# B&R Automation Studio project Snapshot (part 2)

#### Function Description1.txt
```
===================================================================================#
This is a sample trak project for the purposes of testing out the snapshot feature.#
===================================================================================#
Function:                                                                          #
50 shuttles move around the trak to move a product from station to station. This   #
continues until the product is finished and unloaded or rejected and removed.      #
                                                                                   #
                                                                                   #
Production stages:                                                                 #
The product can exist in four different states. At each stage, the product becomes #
harder/firmer and can be moved faster and accelerated quicker. The four stages and #
their respective parameters are:                                                   #
                                                                                   #
1 YELLOW (Liquid)                                                                  #
	veloctiy    = 0.5 m/s                                                          #
	accel/decel = 5 m/s^2                                                          #
	destination = stn 2                                                            #
2 BLUE (Gel)                                                                       #
	veloctiy    = 1 m/s                                                            #
	accel/decel = 10 m/s^2                                                         #
	destination = stn 3                                                            #
3 ORANGE (Soft Solid)                                                              #
	veloctiy    = 2 m/s                                                            #
	accel/decel = 15 m/s^2                                                         #
	destination = stn 4                                                            #
4 GREEN (Solid)                                                                    #
	veloctiy    = 2.5 m/s                                                          #
	accel/decel = 20 m/s^2                                                         #
	destination = stn 1 (offload)                                                  #
                                                                                   #
                                                                                   #
Additional stages:                                                                 #
The two additional stages are:                                                     #
                                                                                   #
1 GRAY (Empty Shuttle)                                                             #
	veloctiy    = 4 m/s                                                            #
	accel/decel = 20 m/s^2                                                         #
	destination = stn 1                                                            #
2 RED (Rejected Product)                                                           #
	veloctiy    = retains speed based on matter state                              #
	accel/decel = retains accel/decel based on matter state                        #
	destination = stn 5 (liquids and gels) or stn 6 (Soft Solids and Solids)       #
                                                                                   #
                                                                                   #
Station Descriptions:                                                              #
                                                                                   #
1 Load/Unload                                                                      #
	Empty shuttles recieve a liquid product                                        #
	GRAY -> YELLOW                                                                 #
	Goes to stn 2                                                                  #
	Finished solid products are removed and the empty shuttles are sent around     #
	GREEN -> GREY                                                                  #
	Goes to stn 1                                                                  #
2 Process 1                                                                        #
	Liquid products are made into gels                                             #
	YELLOW -> BLUE                                                                 #
	Goes to stn 3                                                                  #
3 Process 2                                                                        #
	Gel products are made into soft solids                                         #
	BLUE -> ORANGE                                                                 #
	Goes to stn 4                                                                  #
4 Process 3                                                                        #
	Soft solid products are made into solids                                       #
	ORANGE -> GREEN                                                                #
	Goes to stn 1                                                                  #
5 Reject 1                                                                         #
	Rejected liquid and gel products are removed                                   #
	RED -> GRAY                                                                    #
	Goes to stn 1                                                                  #
6 Reject 2                                                                         #
	Rejected soft solid and solid products are removed                             #
	RED -> GREY                                                                    #
	Goes to stn 1                                                                  #
                                                                                   #
                                                                                   #
At random times, stations will detect rejects, turn them red, and send them to the #
appropriate reject stations.                                                       #
===================================================================================#
```

#### Init.st
```iecst
PROGRAM _INIT
	//Build the array of station references
	Stn[1]  := ADR(Load_Unload_Sector);

	Stn[2]  := ADR(Process_1_Sector);

	Stn[3]  := ADR(Process_2_Sector);

	Stn[4]  := ADR(Process_3_Sector);

	Stn[5]  := ADR(Reject_LeftUp);
	Stn[6]  := ADR(Reject_RightUp);
	Stn[7]  := ADR(Reject_RightDown);

	Stn[8]  := ADR(Flipper_LeftUp);
	Stn[9]  := ADR(Flipper_RightUp);
	Stn[10] := ADR(Flipper_RightDown);

	//List the segment sectors
	SECTOR_SEG_01;
	SECTOR_SEG_02;
	SECTOR_SEG_03;
	SECTOR_SEG_04;
	SECTOR_SEG_05;
	SECTOR_SEG_06;
	SECTOR_SEG_07;
	SECTOR_SEG_08;
	SECTOR_SEG_09;
	SECTOR_SEG_10;
	SECTOR_SEG_11;
	SECTOR_SEG_12;
	SECTOR_SEG_13;
	SECTOR_SEG_14;
	SECTOR_SEG_15;
	SECTOR_SEG_16;
	SECTOR_SEG_17;
	SECTOR_SEG_18;
	SECTOR_SEG_19;
	SECTOR_SEG_20;
	SECTOR_SEG_21;
	SECTOR_SEG_22;
	SECTOR_SEG_23;
	SECTOR_SEG_24;
	SECTOR_SEG_25;
	SECTOR_SEG_26;
	SECTOR_SEG_27;
	SECTOR_SEG_28;
	SECTOR_SEG_29;
	SECTOR_SEG_30;
	SECTOR_SEG_31;
	SECTOR_SEG_32;
	SECTOR_SEG_33;
	SECTOR_SEG_34;
	SECTOR_SEG_35;
	SECTOR_SEG_36;
	SECTOR_SEG_37;
	SECTOR_SEG_38;
	SECTOR_SEG_39;
	SECTOR_SEG_40;
	SECTOR_SEG_41;
	SECTOR_SEG_42;
	SECTOR_SEG_43;
	SECTOR_SEG_44;
	SECTOR_SEG_45;
	SECTOR_SEG_46;
	SECTOR_SEG_47;
	SECTOR_SEG_48;
	SECTOR_SEG_49;
	SECTOR_SEG_50;
	SECTOR_SEG_51;
	SECTOR_SEG_52;
	SECTOR_SEG_53;
	SECTOR_SEG_54;
	SECTOR_SEG_55;
	SECTOR_SEG_56;
	SECTOR_SEG_57;
	SECTOR_SEG_58;
	SECTOR_SEG_59;
	SECTOR_SEG_60;
	SECTOR_SEG_61;
	SECTOR_SEG_62;
	SECTOR_SEG_63;
	SECTOR_SEG_64;
	SECTOR_SEG_65;
	SECTOR_SEG_66;
	SECTOR_SEG_67;
	SECTOR_SEG_68;
	SECTOR_SEG_69;
	SECTOR_SEG_70;
END_PROGRAM
```

#### Main.st
```iecst
PROGRAM _CYCLIC

	BarrierReadInfo.ProcessPoint := ADR(PP_RejectEntrance);
	BarrierReadInfo.Enable       := TRUE;
	BarrierReadInfo();

	CASE TrakState OF
		TRAK_IDLE:
			IF gPowerOn THEN
				AsmPowerOn.Assembly := ADR(gAssembly_1);
				AsmPowerOn.Execute  := TRUE;
				TrakState           := TRAK_POWERON;
			END_IF

		TRAK_POWERON:
			IF AsmPowerOn.Done THEN
				AsmGetShuttle.Assembly := ADR(gAssembly_1);
				AsmGetShuttle.Enable   := TRUE;
				TrakState              := TRAK_FIND_SHUTTLE;   //USE THIS FOR REGULAR OPERATION
//				TrakState              := TRAK_SYSTEM_RUNNING; //USE THIS FOR SPAWNING OPERATION
			END_IF

		TRAK_FIND_SHUTTLE:
			IF AsmGetShuttle.Valid THEN
				AsmData.Color                 := GRAY;
				AsmCopyUserData.Axis          := ADR(AsmGetShuttle.Axis);
				AsmCopyUserData.DataAddress   := ADR(AsmData);
				AsmCopyUserData.DataSize      := SIZEOF(AsmData);
				AsmCopyUserData.Mode          := mcACPTRAK_USERDATA_SET;
				AsmCopyUserData.Execute       := TRUE;

				AsmGetShuttle.Next            := FALSE;
				AsmRoutedMoveAbs.Axis         := ADR(AsmGetShuttle.Axis);
				AsmRoutedMoveAbs.Sector       := Stn[1];
				AsmRoutedMoveAbs.Position     := 0.005;
				AsmRoutedMoveAbs.Acceleration := 20;
				AsmRoutedMoveAbs.Deceleration := 20;
				AsmRoutedMoveAbs.Velocity     := 4;
				AsmRoutedMoveAbs.Execute      := TRUE;

				TrakState                     := TRAK_SEND_SHUTTLE;
			END_IF

		TRAK_SEND_SHUTTLE:
			IF AsmRoutedMoveAbs.Active AND AsmCopyUserData.Done THEN
				IF (AsmGetShuttle.RemainingCount > 0) THEN
					AsmCopyUserData.Execute  := FALSE;
					AsmRoutedMoveAbs.Execute := FALSE;
					AsmGetShuttle.Next       := TRUE;
					//AsmIndex               := AsmIndex + 1;
					TrakState                := TRAK_FIND_SHUTTLE;
				ELSE
					AsmGetShuttle.Enable := FALSE;
					gTrakRunning         := TRUE;
					TrakState            := TRAK_SYSTEM_RUNNING;
				END_IF
			END_IF

		TRAK_SYSTEM_RUNNING:

	END_CASE

	//Call FUBs
	AsmPowerOn();
	AsmGetShuttle();
	AsmCopyUserData();
	AsmRoutedMoveAbs();

	//Call action files
	Load_Unload;
	Process_1;
	Process_2;
	Process_3;
	Reject;
	RejectExit;
	Flipper;
	FlipperExit;

END_PROGRAM
```

#### 1_Load_Unload.st
```iecst
ACTION Load_Unload:

	TrgPointEnable[1].ProcessPoint  := ADR(PP_Load_Unload);
	TrgPointEnable[1].Enable        := TRUE;
	TrgPointGetInfo[1].ProcessPoint := ADR(PP_Load_Unload);

	CASE StnState[1] OF
		STN_WAIT_FOR_SHUTTLE:
			IF (TrgPointEnable[1].EventCount > 0) THEN
				TrgPointGetInfo[1].Execute := TRUE;
				StnState[1]                := STN_GET_INFO;
			END_IF

		STN_GET_INFO:
			IF TrgPointGetInfo[1].Done THEN
				ShCopyUserData[1].Axis        := ADR(TrgPointGetInfo[1].TrgPointInfo.Axis);
				ShCopyUserData[1].DataAddress := ADR(StationData[1]);
				ShCopyUserData[1].DataSize    := SIZEOF(StationData[1]);
				ShCopyUserData[1].Mode        := mcACPTRAK_USERDATA_GET;
				ShCopyUserData[1].Execute     := TRUE;
				StnState[1]                   := STN_GET_USERDATA;
			END_IF

		STN_GET_USERDATA:
			IF ShCopyUserData[1].Done THEN
				ShCopyUserData[1].Execute := FALSE;
				IF (StationData[1].Color = GRAY) OR (StationData[1].Color = GREEN) THEN
					StnState[1] := STN_HANDLE_SHUTTLE;
				ELSE
					TrgPointGetInfo[1].Execute := FALSE;
					StnState[1]                := STN_WAIT_FOR_SHUTTLE;
				END_IF
			END_IF

		STN_HANDLE_SHUTTLE:
			IF (StationData[1].Color = GRAY) THEN
				StationData[1].Color                                      := YELLOW;
				StnRoutedMoveAbs[1].Axis                                  := ADR(TrgPointGetInfo[1].TrgPointInfo.Axis);
				StnRoutedMoveAbs[1].Sector                                := Stn[2];
				StnRoutedMoveAbs[1].Position                              := 0.005;
				StnRoutedMoveAbs[1].Acceleration                          := 5;
				StnRoutedMoveAbs[1].Deceleration                          := 5;
				StnRoutedMoveAbs[1].Velocity                              := 0.5;
				StnRoutedMoveAbs[5].AdvancedParameters.ShuttleOrientation := mcDIR_UNDEFINED;
				StnRoutedMoveAbs[1].AdvancedParameters.StartDirection     := mcDIR_POSITIVE;
				StnRoutedMoveAbs[1].AdvancedParameters.EndDirection       := mcDIR_POSITIVE;
			ELSIF (StationData[1].Color = GREEN) THEN
				IF (RejectIndex[1] = RejectRate) THEN
					StationData[1].Color                                      := RED;
					StnRoutedMoveAbs[1].Axis                                  := ADR(TrgPointGetInfo[1].TrgPointInfo.Axis);
					StnRoutedMoveAbs[1].Sector                                := Stn[6];
					StnRoutedMoveAbs[1].Position                              := 0.405;
					StnRoutedMoveAbs[1].Acceleration                          := 20;
					StnRoutedMoveAbs[1].Deceleration                          := 20;
					StnRoutedMoveAbs[1].Velocity                              := 2.5;
					StnRoutedMoveAbs[1].AdvancedParameters.ShuttleOrientation := mcDIR_UNDEFINED;
					StnRoutedMoveAbs[1].AdvancedParameters.StartDirection     := mcDIR_POSITIVE;
					StnRoutedMoveAbs[1].AdvancedParameters.EndDirection       := mcDIR_POSITIVE;
					RejectIndex[1]                                            := 0;
				ELSE
					StationData[1].Color := GRAY;
					StnRoutedMoveAbs[1].Axis                                  := ADR(TrgPointGetInfo[1].TrgPointInfo.Axis);
					StnRoutedMoveAbs[1].Sector                                := Stn[1];
					StnRoutedMoveAbs[1].Position                              := 0.004;
					StnRoutedMoveAbs[1].Acceleration                          := 20;
					StnRoutedMoveAbs[1].Deceleration                          := 20;
					StnRoutedMoveAbs[1].Velocity                              := 4;
					StnRoutedMoveAbs[5].AdvancedParameters.ShuttleOrientation := mcDIR_UNDEFINED;
					StnRoutedMoveAbs[1].AdvancedParameters.StartDirection     := mcDIR_POSITIVE;
					StnRoutedMoveAbs[1].AdvancedParameters.EndDirection       := mcDIR_POSITIVE;
					RejectIndex[1]                                            := RejectIndex[1] + 1;
				END_IF
			END_IF
			ShCopyUserData[1].Mode    := mcACPTRAK_USERDATA_SET;
			ShCopyUserData[1].Execute := TRUE;
			StnState[1]               := STN_SET_USERDATA;

		STN_SET_USERDATA:
			IF ShCopyUserData[1].Done THEN
				ShCopyUserData[1].Execute   := FALSE;
				StnRoutedMoveAbs[1].Execute := TRUE;
				StnState[1]                 := STN_SEND_SHUTTLE;
			END_IF

		STN_SEND_SHUTTLE:
			IF StnRoutedMoveAbs[1].Active THEN
				TrgPointGetInfo[1].Execute  := FALSE;
				StnRoutedMoveAbs[1].Execute := FALSE;
				StnState[1]                 := STN_WAIT_FOR_SHUTTLE;
			END_IF

	END_CASE

	TrgPointEnable[1]();
	TrgPointGetInfo[1]();
	ShCopyUserData[1]();
	StnRoutedMoveAbs[1]();

END_ACTION
```

#### 2_Process_1.st
```iecst
ACTION Process_1:

	TrgPointEnable[2].ProcessPoint  := ADR(PP_Process_1);
	TrgPointEnable[2].Enable        := TRUE;
	TrgPointGetInfo[2].ProcessPoint := ADR(PP_Process_1);

	CASE StnState[2] OF
		STN_WAIT_FOR_SHUTTLE:
			IF (TrgPointEnable[2].EventCount > 0) THEN
				TrgPointGetInfo[2].Execute := TRUE;
				StnState[2]                := STN_GET_INFO;
			END_IF

		STN_GET_INFO:
			IF TrgPointGetInfo[2].Done THEN
				ShCopyUserData[2].Axis        := ADR(TrgPointGetInfo[2].TrgPointInfo.Axis);
				ShCopyUserData[2].DataAddress := ADR(StationData[2]);
				ShCopyUserData[2].DataSize    := SIZEOF(StationData[2]);
				ShCopyUserData[2].Mode        := mcACPTRAK_USERDATA_GET;
				ShCopyUserData[2].Execute     := TRUE;
				StnState[2]                   := STN_GET_USERDATA;
			END_IF

		STN_GET_USERDATA:
			IF ShCopyUserData[2].Done THEN
				ShCopyUserData[2].Execute := FALSE;
				IF (StationData[2].Color = YELLOW) THEN
					StnState[2] := STN_HANDLE_SHUTTLE;
				ELSE
					TrgPointGetInfo[2].Execute := FALSE;
					StnState[2]                := STN_WAIT_FOR_SHUTTLE;
				END_IF
			END_IF

		STN_HANDLE_SHUTTLE:
			IF (StationData[2].Color = YELLOW) THEN
				IF (RejectIndex[2] = RejectRate) THEN
					StationData[2].Color                                      := RED;
					StnRoutedMoveAbs[2].Axis                                  := ADR(TrgPointGetInfo[2].TrgPointInfo.Axis);
					StnRoutedMoveAbs[2].Sector                                := Stn[6];
					StnRoutedMoveAbs[2].Position                              := 0.405;
					StnRoutedMoveAbs[2].Acceleration                          := 5;
					StnRoutedMoveAbs[2].Deceleration                          := 5;
					StnRoutedMoveAbs[2].Velocity                              := 0.5;
					StnRoutedMoveAbs[5].AdvancedParameters.ShuttleOrientation := mcDIR_UNDEFINED;
					StnRoutedMoveAbs[2].AdvancedParameters.StartDirection     := mcDIR_POSITIVE;
					StnRoutedMoveAbs[2].AdvancedParameters.EndDirection       := mcDIR_POSITIVE;
					RejectIndex[2]                                            := 0;
				ELSE
					StationData[2].Color                                      := BLUE;
					StnRoutedMoveAbs[2].Axis                                  := ADR(TrgPointGetInfo[2].TrgPointInfo.Axis);
					StnRoutedMoveAbs[2].Sector                                := Stn[3];
					StnRoutedMoveAbs[2].Position                              := 0.005;
					StnRoutedMoveAbs[2].Acceleration                          := 10;
					StnRoutedMoveAbs[2].Deceleration                          := 10;
					StnRoutedMoveAbs[2].Velocity                              := 1;
					StnRoutedMoveAbs[5].AdvancedParameters.ShuttleOrientation := mcDIR_UNDEFINED;
					StnRoutedMoveAbs[2].AdvancedParameters.StartDirection     := mcDIR_POSITIVE;
					StnRoutedMoveAbs[2].AdvancedParameters.EndDirection       := mcDIR_POSITIVE;
					RejectIndex[2]                                            := RejectIndex[2] + 1;
				END_IF
			END_IF
			ShCopyUserData[2].Mode    := mcACPTRAK_USERDATA_SET;
			ShCopyUserData[2].Execute := TRUE;
			StnState[2]               := STN_SET_USERDATA;

		STN_SET_USERDATA:
			IF ShCopyUserData[2].Done THEN
				ShCopyUserData[2].Execute   := FALSE;
				StnRoutedMoveAbs[2].Execute := TRUE;
				StnState[2]                 := STN_SEND_SHUTTLE;
			END_IF

		STN_SEND_SHUTTLE:
			IF StnRoutedMoveAbs[2].Active THEN
				TrgPointGetInfo[2].Execute  := FALSE;
				StnRoutedMoveAbs[2].Execute := FALSE;
				StnState[2]                 := STN_WAIT_FOR_SHUTTLE;
			END_IF

	END_CASE

	TrgPointEnable[2]();
	TrgPointGetInfo[2]();
	ShCopyUserData[2]();
	StnRoutedMoveAbs[2]();

END_ACTION
```

#### 3_Process_2.st
```iecst
ACTION Process_2:

	TrgPointEnable[3].ProcessPoint  := ADR(PP_Process_2);
	TrgPointEnable[3].Enable        := TRUE;
	TrgPointGetInfo[3].ProcessPoint := ADR(PP_Process_2);

	CASE StnState[3] OF
		STN_WAIT_FOR_SHUTTLE:
			IF (TrgPointEnable[3].EventCount > 0) THEN
				TrgPointGetInfo[3].Execute := TRUE;
				StnState[3]                := STN_GET_INFO;
			END_IF

		STN_GET_INFO:
			IF TrgPointGetInfo[3].Done THEN
				ShCopyUserData[3].Axis        := ADR(TrgPointGetInfo[3].TrgPointInfo.Axis);
				ShCopyUserData[3].DataAddress := ADR(StationData[3]);
				ShCopyUserData[3].DataSize    := SIZEOF(StationData[3]);
				ShCopyUserData[3].Mode        := mcACPTRAK_USERDATA_GET;
				ShCopyUserData[3].Execute     := TRUE;
				StnState[3]                   := STN_GET_USERDATA;
			END_IF

		STN_GET_USERDATA:
			IF ShCopyUserData[3].Done THEN
				ShCopyUserData[3].Execute := FALSE;
				IF (StationData[3].Color = BLUE) THEN
					StnState[3] := STN_HANDLE_SHUTTLE;
				ELSE
					TrgPointGetInfo[3].Execute := FALSE;
					StnState[3]                := STN_WAIT_FOR_SHUTTLE;
				END_IF
			END_IF

		STN_HANDLE_SHUTTLE:
			IF (StationData[3].Color = BLUE) THEN
				IF (RejectIndex[3] = RejectRate) THEN
					StationData[3].Color                                      := RED;
					StnRoutedMoveAbs[3].Axis                                  := ADR(TrgPointGetInfo[3].TrgPointInfo.Axis);
					StnRoutedMoveAbs[3].Sector                                := Stn[6];
					StnRoutedMoveAbs[3].Position                              := 0.405;
					StnRoutedMoveAbs[3].Acceleration                          := 10;
					StnRoutedMoveAbs[3].Deceleration                          := 10;
					StnRoutedMoveAbs[3].Velocity                              := 1;
					StnRoutedMoveAbs[3].AdvancedParameters.ShuttleOrientation := mcDIR_UNDEFINED;
					StnRoutedMoveAbs[3].AdvancedParameters.StartDirection     := mcDIR_POSITIVE;
					StnRoutedMoveAbs[3].AdvancedParameters.EndDirection       := mcDIR_POSITIVE;
					RejectIndex[3]                                            := 0;
				ELSE
					StationData[3].Color                                      := ORANGE;
					StnRoutedMoveAbs[3].Axis                                  := ADR(TrgPointGetInfo[3].TrgPointInfo.Axis);
					StnRoutedMoveAbs[3].Sector                                := Stn[4];
					StnRoutedMoveAbs[3].Position                              := 0.005;
					StnRoutedMoveAbs[3].Acceleration                          := 15;
					StnRoutedMoveAbs[3].Deceleration                          := 15;
					StnRoutedMoveAbs[3].Velocity                              := 2;
					StnRoutedMoveAbs[5].AdvancedParameters.ShuttleOrientation := mcDIR_UNDEFINED;
					StnRoutedMoveAbs[3].AdvancedParameters.StartDirection     := mcDIR_POSITIVE;
					StnRoutedMoveAbs[3].AdvancedParameters.EndDirection       := mcDIR_POSITIVE;
					RejectIndex[3]                                            := RejectIndex[3] + 1;
				END_IF
			END_IF
			ShCopyUserData[3].Mode    := mcACPTRAK_USERDATA_SET;
			ShCopyUserData[3].Execute := TRUE;
			StnState[3]               := STN_SET_USERDATA;

		STN_SET_USERDATA:
			IF ShCopyUserData[3].Done THEN
				ShCopyUserData[3].Execute   := FALSE;
				StnRoutedMoveAbs[3].Execute := TRUE;
				StnState[3]                 := STN_SEND_SHUTTLE;
			END_IF

		STN_SEND_SHUTTLE:
			IF StnRoutedMoveAbs[3].Active THEN
				TrgPointGetInfo[3].Execute  := FALSE;
				StnRoutedMoveAbs[3].Execute := FALSE;
				StnState[3]                 := STN_WAIT_FOR_SHUTTLE;
			END_IF

	END_CASE

	TrgPointEnable[3]();
	TrgPointGetInfo[3]();
	ShCopyUserData[3]();
	StnRoutedMoveAbs[3]();

END_ACTION
```

#### 4_Process_3.st
```iecst
ACTION Process_3:

	TrgPointEnable[4].ProcessPoint  := ADR(PP_Process_3);
	TrgPointEnable[4].Enable        := TRUE;
	TrgPointGetInfo[4].ProcessPoint := ADR(PP_Process_3);

	CASE StnState[4] OF
		STN_WAIT_FOR_SHUTTLE:
			IF (TrgPointEnable[4].EventCount > 0) THEN
				TrgPointGetInfo[4].Execute := TRUE;
				StnState[4]                := STN_GET_INFO;
			END_IF

		STN_GET_INFO:
			IF TrgPointGetInfo[4].Done THEN
				ShCopyUserData[4].Axis        := ADR(TrgPointGetInfo[4].TrgPointInfo.Axis);
				ShCopyUserData[4].DataAddress := ADR(StationData[4]);
				ShCopyUserData[4].DataSize    := SIZEOF(StationData[4]);
				ShCopyUserData[4].Mode        := mcACPTRAK_USERDATA_GET;
				ShCopyUserData[4].Execute     := TRUE;
				StnState[4]                   := STN_GET_USERDATA;
			END_IF

		STN_GET_USERDATA:
			IF ShCopyUserData[4].Done THEN
				ShCopyUserData[4].Execute := FALSE;
				IF (StationData[4].Color = ORANGE) THEN
					StnState[4] := STN_HANDLE_SHUTTLE;
				ELSE
					TrgPointGetInfo[4].Execute := FALSE;
					StnState[4]                := STN_WAIT_FOR_SHUTTLE;
				END_IF
			END_IF

		STN_HANDLE_SHUTTLE:
			IF (StationData[4].Color = ORANGE) THEN
				IF (RejectIndex[4] = RejectRate) THEN
					StationData[4].Color                                      := RED;
					StnRoutedMoveAbs[4].Axis                                  := ADR(TrgPointGetInfo[4].TrgPointInfo.Axis);
					StnRoutedMoveAbs[4].Sector                                := Stn[6];
					StnRoutedMoveAbs[4].Position                              := 0.405;
					StnRoutedMoveAbs[4].Acceleration                          := 15;
					StnRoutedMoveAbs[4].Deceleration                          := 15;
					StnRoutedMoveAbs[4].Velocity                              := 2;
					StnRoutedMoveAbs[4].AdvancedParameters.ShuttleOrientation := mcDIR_UNDEFINED;
					StnRoutedMoveAbs[4].AdvancedParameters.StartDirection     := mcDIR_POSITIVE;
					StnRoutedMoveAbs[4].AdvancedParameters.EndDirection       := mcDIR_POSITIVE;
					RejectIndex[4]                                            := 0;
				ELSE
					StationData[4].Color                                      := GREEN;
					StnRoutedMoveAbs[4].Axis                                  := ADR(TrgPointGetInfo[4].TrgPointInfo.Axis);
					StnRoutedMoveAbs[4].Sector                                := Stn[1];
					StnRoutedMoveAbs[4].Position                              := 0.005;
					StnRoutedMoveAbs[4].Acceleration                          := 20;
					StnRoutedMoveAbs[4].Deceleration                          := 20;
					StnRoutedMoveAbs[4].Velocity                              := 2.5;
					StnRoutedMoveAbs[5].AdvancedParameters.ShuttleOrientation := mcDIR_UNDEFINED;
					StnRoutedMoveAbs[4].AdvancedParameters.StartDirection     := mcDIR_POSITIVE;
					StnRoutedMoveAbs[4].AdvancedParameters.EndDirection       := mcDIR_POSITIVE;
					RejectIndex[4]                                            := RejectIndex[4] + 1;
				END_IF
			END_IF
			ShCopyUserData[4].Mode    := mcACPTRAK_USERDATA_SET;
			ShCopyUserData[4].Execute := TRUE;
			StnState[4]               := STN_SET_USERDATA;

		STN_SET_USERDATA:
			IF ShCopyUserData[4].Done THEN
				ShCopyUserData[4].Execute   := FALSE;
				StnRoutedMoveAbs[4].Execute := TRUE;
				StnState[4]                 := STN_SEND_SHUTTLE;
			END_IF

		STN_SEND_SHUTTLE:
			IF StnRoutedMoveAbs[4].Active THEN
				TrgPointGetInfo[4].Execute  := FALSE;
				StnRoutedMoveAbs[4].Execute := FALSE;
				StnState[4]                 := STN_WAIT_FOR_SHUTTLE;
			END_IF

	END_CASE

	TrgPointEnable[4]();
	TrgPointGetInfo[4]();
	ShCopyUserData[4]();
	StnRoutedMoveAbs[4]();

END_ACTION
```

#### 6_Reject.st
```iecst
ACTION Reject:

	TrgPointEnable[5].ProcessPoint  := ADR(PP_Reject);
	TrgPointEnable[5].Enable        := TRUE;
	TrgPointGetInfo[5].ProcessPoint := ADR(PP_Reject);

	CASE StnState[5] OF
		STN_WAIT_FOR_SHUTTLE:
			IF (TrgPointEnable[5].EventCount > 0) THEN
				TrgPointGetInfo[5].Execute := TRUE;
				StnState[5]                := STN_GET_INFO;
			END_IF

		STN_GET_INFO:
			IF TrgPointGetInfo[5].Done THEN
				ShReadInfo[5].Axis            := ADR(TrgPointGetInfo[5].TrgPointInfo.Axis);
				ShReadInfo[5].Enable          := TRUE;
				ShCopyUserData[5].Axis        := ADR(TrgPointGetInfo[5].TrgPointInfo.Axis);
				ShCopyUserData[5].DataAddress := ADR(StationData[5]);
				ShCopyUserData[5].DataSize    := SIZEOF(StationData[5]);
				ShCopyUserData[5].Mode        := mcACPTRAK_USERDATA_GET;
				ShCopyUserData[5].Execute     := TRUE;
				StnState[5]                   := STN_GET_USERDATA;
			END_IF

		STN_GET_USERDATA:
			IF ShCopyUserData[5].Done AND (ShReadInfo[5].ShuttleInfo.AdditionalInfo.PLCopenState = mcAXIS_STANDSTILL) THEN
				ShCopyUserData[5].Execute := FALSE;
				IF (StationData[5].Color = RED) THEN
					ShSwitchSector[5].Axis    := ADR(TrgPointGetInfo[5].TrgPointInfo.Axis);
					ShSwitchSector[5].Sector  := Stn[7];
					ShSwitchSector[5].Execute := TRUE;
					StnState[5]               := STN_HANDLE_SHUTTLE;
				ELSE
					TrgPointGetInfo[5].Execute := FALSE;
					ShReadInfo[5].Enable       := FALSE;
					StnState[5]                := STN_WAIT_FOR_SHUTTLE;
				END_IF
			END_IF

		STN_HANDLE_SHUTTLE:
			IF (ShSwitchSector[5].Done) AND (ShReadInfo[5].ShuttleInfo.CurrentValues.SectorName = 'Reject_RightDown') THEN
				ShSwitchSector[5].Execute                                 := FALSE;
				StationData[5].Color                                      := GRAY;
				StnRoutedMoveAbs[5].Axis                                  := ADR(TrgPointGetInfo[5].TrgPointInfo.Axis);
				StnRoutedMoveAbs[5].Sector                                := Stn[9];
				StnRoutedMoveAbs[5].Position                              := 0.405;
				StnRoutedMoveAbs[5].Acceleration                          := 20;
				StnRoutedMoveAbs[5].Deceleration                          := 20;
				StnRoutedMoveAbs[5].Velocity                              := 4;
				StnRoutedMoveAbs[5].AdvancedParameters.ShuttleOrientation := mcDIR_UNDEFINED;
				StnRoutedMoveAbs[5].AdvancedParameters.StartDirection     := mcDIR_POSITIVE;
				StnRoutedMoveAbs[5].AdvancedParameters.EndDirection       := mcDIR_POSITIVE;
				ShCopyUserData[5].Mode                                    := mcACPTRAK_USERDATA_SET;
				ShCopyUserData[5].Execute                                 := TRUE;
				StnState[5]                                               := STN_SET_USERDATA;
			END_IF

		STN_SET_USERDATA:
			IF ShCopyUserData[5].Done THEN
				ShCopyUserData[5].Execute   := FALSE;
				StnRoutedMoveAbs[5].Execute := TRUE;
				StnState[5]                 := STN_SEND_SHUTTLE;
			END_IF

		STN_SEND_SHUTTLE:
			IF StnRoutedMoveAbs[5].Active THEN
				TrgPointGetInfo[5].Execute  := FALSE;
				ShReadInfo[5].Enable        := FALSE;
				StnRoutedMoveAbs[5].Execute := FALSE;
				StnState[5]                 := STN_WAIT_FOR_SHUTTLE;
			END_IF

	END_CASE

	TrgPointEnable[5]();
	TrgPointGetInfo[5]();
	ShCopyUserData[5]();
	ShReadInfo[5]();
	ShSwitchSector[5]();
	StnRoutedMoveAbs[5]();

END_ACTION
```

#### 6_RejectEntrance.st
```iecst
ACTION RejectEntrance:

END_ACTION
```

#### 6_RejectExit.st
```iecst
ACTION RejectExit:

	GateTrgPointEnable[0].ProcessPoint := ADR(PP_RejectExit);
	GateTrgPointEnable[0].Enable       := TRUE;

	GateTrgPointGetInfo[0].ProcessPoint := ADR(PP_RejectExit);

	GateBarrierCommand[0].ProcessPoint                   := ADR(PP_RejectEntrance);
	GateBarrierCommand[0].AdvancedParameters.TicketCount := 1;

	CASE ExitState[0] OF

		EXIT_INIT:
			IF NOT GateInit[0] THEN
				GateBarrierCommand[0].Command := mcACPTRAK_BARRIER_CLOSE;
				GateBarrierCommand[0].Execute := TRUE;
				GateInit[0]                   := TRUE;
			ELSIF GateInit[0] AND GateBarrierCommand[0].Done THEN
				GateBarrierCommand[0].Execute := FALSE;
			ELSIF GateInit[0] AND NOT GateBarrierCommand[0].Execute THEN
				GateBarrierCommand[0].Command := mcACPTRAK_BARRIER_ADD_TICKETS;
				GateBarrierCommand[0].Execute := TRUE;
				ExitState[0]                  := EXIT_WAIT_FOR_SHUTTLE;
			END_IF

		EXIT_WAIT_FOR_SHUTTLE:
			IF GateBarrierCommand[0].Done THEN
				GateBarrierCommand[0].Execute := FALSE;
			END_IF

			IF (GateTrgPointEnable[0].EventCount > 0) THEN
				GateTrgPointGetInfo[0].Execute := TRUE;
				ExitState[0]                   := EXIT_GET_INFO;
			END_IF

		EXIT_GET_INFO:
			IF GateTrgPointGetInfo[0].Done THEN
				GateTrgPointGetInfo[0].Execute := FALSE;
				GateBarrierCommand[0].Execute  := TRUE;
				ExitState[0]                   := EXIT_GIVE_TICKET;
			END_IF

		EXIT_GIVE_TICKET:
			IF GateBarrierCommand[0].Done THEN
				GateBarrierCommand[0].Execute := FALSE;
				Temp_NumTickets               := Temp_NumTickets + 1;
				ExitState[0]                  := EXIT_WAIT_FOR_SHUTTLE;
			END_IF

	END_CASE

	//FUB Calls
	GateTrgPointEnable[0]();
	GateTrgPointGetInfo[0]();
	GateBarrierCommand[0]();

END_ACTION
```

#### 9_Flipper.st
```iecst
ACTION Flipper:

	TrgPointEnable[6].ProcessPoint  := ADR(PP_Flipper);
	TrgPointEnable[6].Enable        := TRUE;
	TrgPointGetInfo[6].ProcessPoint := ADR(PP_Flipper);

	CASE StnState[6] OF
		STN_WAIT_FOR_SHUTTLE:
			IF (TrgPointEnable[6].EventCount > 0) THEN
				TrgPointGetInfo[6].Execute := TRUE;
				StnState[6]                := STN_GET_INFO;
			END_IF

		STN_GET_INFO:
			IF TrgPointGetInfo[6].Done THEN
				ShReadInfo[6].Axis            := ADR(TrgPointGetInfo[6].TrgPointInfo.Axis);
				ShReadInfo[6].Enable          := TRUE;
				ShCopyUserData[6].Axis        := ADR(TrgPointGetInfo[6].TrgPointInfo.Axis);
				ShCopyUserData[6].DataAddress := ADR(StationData[6]);
				ShCopyUserData[6].DataSize    := SIZEOF(StationData[6]);
				ShCopyUserData[6].Mode        := mcACPTRAK_USERDATA_GET;
				ShCopyUserData[6].Execute     := TRUE;
				StnState[6]                   := STN_GET_USERDATA;
			END_IF

		STN_GET_USERDATA:
			IF ShCopyUserData[6].Done AND (ShReadInfo[6].ShuttleInfo.AdditionalInfo.PLCopenState = mcAXIS_STANDSTILL) THEN
				ShCopyUserData[6].Execute := FALSE;
				IF (StationData[6].Color = GRAY) THEN
					ShSwitchSector[6].Axis    := ADR(TrgPointGetInfo[6].TrgPointInfo.Axis);
					ShSwitchSector[6].Sector  := Stn[10];
					ShSwitchSector[6].Execute := TRUE;
					StnState[6]               := STN_HANDLE_SHUTTLE;
				ELSE
					TrgPointGetInfo[6].Execute := FALSE;
					ShReadInfo[6].Enable       := FALSE;
					StnState[6]                := STN_WAIT_FOR_SHUTTLE;
				END_IF
			END_IF

		STN_HANDLE_SHUTTLE:
			IF (ShSwitchSector[6].Done) AND (ShReadInfo[6].ShuttleInfo.CurrentValues.SectorName = 'Flipper_RightDown') THEN
				ShSwitchSector[6].Execute                                 := FALSE;
				StationData[6].Color                                      := GRAY;
				StnRoutedMoveAbs[6].Axis                                  := ADR(TrgPointGetInfo[6].TrgPointInfo.Axis);
				StnRoutedMoveAbs[6].Sector                                := Stn[1];
				StnRoutedMoveAbs[6].Position                              := 0.005;
				StnRoutedMoveAbs[6].Acceleration                          := 20;
				StnRoutedMoveAbs[6].Deceleration                          := 20;
				StnRoutedMoveAbs[6].Velocity                              := 4;
				StnRoutedMoveAbs[6].AdvancedParameters.ShuttleOrientation := mcDIR_UNDEFINED;
				StnRoutedMoveAbs[6].AdvancedParameters.StartDirection     := mcDIR_POSITIVE;
				StnRoutedMoveAbs[6].AdvancedParameters.EndDirection       := mcDIR_POSITIVE;
				ShCopyUserData[6].Mode                                    := mcACPTRAK_USERDATA_SET;
				ShCopyUserData[6].Execute                                 := TRUE;
				StnState[6]                                               := STN_SET_USERDATA;
			END_IF

		STN_SET_USERDATA:
			IF ShCopyUserData[6].Done THEN
				ShCopyUserData[6].Execute   := FALSE;
				StnRoutedMoveAbs[6].Execute := TRUE;
				StnState[6]                 := STN_SEND_SHUTTLE;
			END_IF

		STN_SEND_SHUTTLE:
			IF StnRoutedMoveAbs[6].Active THEN
				TrgPointGetInfo[6].Execute  := FALSE;
				ShReadInfo[6].Enable        := FALSE;
				StnRoutedMoveAbs[6].Execute := FALSE;
				StnState[6]                 := STN_WAIT_FOR_SHUTTLE;
			END_IF

	END_CASE

	TrgPointEnable[6]();
	TrgPointGetInfo[6]();
	ShCopyUserData[6]();
	ShReadInfo[6]();
	ShSwitchSector[6]();
	StnRoutedMoveAbs[6]();

END_ACTION
```

#### 9_FlipperEntrance.st
```iecst
ACTION FlipperEntrance:

END_ACTION
```

#### 9_FlipperExit.st
```iecst
ACTION FlipperExit:

	GateTrgPointEnable[1].ProcessPoint := ADR(PP_FlipperExit);
	GateTrgPointEnable[1].Enable       := TRUE;

	GateTrgPointGetInfo[1].ProcessPoint := ADR(PP_FlipperExit);

	GateBarrierCommand[1].ProcessPoint                   := ADR(PP_FlipperEntrance);
	GateBarrierCommand[1].AdvancedParameters.TicketCount := 1;
	GateBarrierCommand[1].Command                        := mcACPTRAK_BARRIER_ADD_TICKETS;

	CASE ExitState[1] OF

		EXIT_INIT:
			IF NOT GateInit[1] THEN
				GateBarrierCommand[1].Command := mcACPTRAK_BARRIER_CLOSE;
				GateBarrierCommand[1].Execute := TRUE;
				GateInit[1]                   := TRUE;
			ELSIF GateInit[1] AND GateBarrierCommand[1].Done THEN
				GateBarrierCommand[1].Execute := FALSE;
			ELSIF GateInit[1] AND NOT GateBarrierCommand[1].Execute THEN
				GateBarrierCommand[1].Command := mcACPTRAK_BARRIER_ADD_TICKETS;
				GateBarrierCommand[1].Execute := TRUE;
				ExitState[1]                  := EXIT_WAIT_FOR_SHUTTLE;
			END_IF

		EXIT_WAIT_FOR_SHUTTLE:
			IF GateBarrierCommand[1].Done THEN
				GateBarrierCommand[1].Execute := FALSE;
			END_IF

			IF (GateTrgPointEnable[1].EventCount > 0) THEN
				GateTrgPointGetInfo[1].Execute := TRUE;
				ExitState[1]                   := EXIT_GET_INFO;
			END_IF

		EXIT_GET_INFO:
			IF GateTrgPointGetInfo[1].Done THEN
				GateTrgPointGetInfo[1].Execute := FALSE;
				GateBarrierCommand[1].Execute  := TRUE;
				ExitState[1]                   := EXIT_GIVE_TICKET;
			END_IF

		EXIT_GIVE_TICKET:
			IF GateBarrierCommand[1].Done THEN
				GateBarrierCommand[1].Execute := FALSE;
				ExitState[1]                  := EXIT_WAIT_FOR_SHUTTLE;
			END_IF

	END_CASE

	//FUB Calls
	GateTrgPointEnable[1]();
	GateTrgPointGetInfo[1]();
	GateBarrierCommand[1]();

END_ACTION
```

#### Types.typ - Local data types
```iecst
TYPE
	TrakState_enum :
		(
		TRAK_IDLE,
		TRAK_POWERON,
		TRAK_FIND_SHUTTLE,
		TRAK_SEND_SHUTTLE,
		TRAK_SYSTEM_RUNNING
		);
	StnState_enum :
		(
		STN_WAIT_FOR_SHUTTLE,
		STN_GET_INFO,
		STN_GET_USERDATA,
		STN_HANDLE_SHUTTLE,
		STN_SET_USERDATA,
		STN_SEND_SHUTTLE
		);
	ExitState_enum :
		(
		EXIT_INIT,
		EXIT_WAIT_FOR_SHUTTLE,
		EXIT_GET_INFO,
		EXIT_GIVE_TICKET
		);
END_TYPE
```

#### Variables.var - Local variables
```iecst
VAR
	BarrierReadInfo : MC_BR_BarrierReadInfo_AcpTrak;
END_VAR
(**)
(*Used in startup*)
VAR
	TrakState : TrakState_enum;
	AsmPowerOn : MC_BR_AsmPowerOn_AcpTrak;
	AsmGetShuttle : MC_BR_AsmGetShuttle_AcpTrak;
	AsmData : UserDataTyp;
	AsmCopyUserData : MC_BR_ShCopyUserData_AcpTrak;
	AsmRoutedMoveAbs : MC_BR_RoutedMoveAbs_AcpTrak;
	AsmIndex : UINT;
	i : UINT;
END_VAR
(**)
(*Used in stations*)
VAR
	Stn : ARRAY[1..10] OF UDINT;
	StnState : ARRAY[1..6] OF StnState_enum;
	TrgPointEnable : ARRAY[1..6] OF MC_BR_TrgPointEnable_AcpTrak;
	TrgPointGetInfo : ARRAY[1..6] OF MC_BR_TrgPointGetInfo_AcpTrak;
	StationData : ARRAY[1..6] OF UserDataTyp;
	ShCopyUserData : ARRAY[1..6] OF MC_BR_ShCopyUserData_AcpTrak;
	StnRoutedMoveAbs : ARRAY[1..6] OF MC_BR_RoutedMoveAbs_AcpTrak;
	ShReadInfo : ARRAY[5..6] OF MC_BR_ShReadInfo_AcpTrak;
	ShSwitchSector : ARRAY[5..6] OF MC_BR_ShSwitchSector_AcpTrak;
	RejectIndex : ARRAY[1..6] OF USINT;
	RejectRate : USINT := 15; (*Every n-th product willl be a reject*)
END_VAR
(**)
(*UsedInGates*)
VAR
	ExitState : ARRAY[0..1] OF ExitState_enum;
	GateTrgPointEnable : ARRAY[0..1] OF MC_BR_TrgPointEnable_AcpTrak;
	GateTrgPointGetInfo : ARRAY[0..1] OF MC_BR_TrgPointGetInfo_AcpTrak;
	GateBarrierCommand : ARRAY[0..1] OF MC_BR_BarrierCommand_AcpTrak;
	GateInit : ARRAY[0..1] OF BOOL;
	Temp_NumTickets : USINT;
END_VAR
```

### Program Logical/SV_Comms (IEC)

#### Variables.var
```iecst
VAR
	Vis : McAcpTrakAssemblyVisData;
	SizeofVis : UDINT := 0;
	NumVisShuttle : USINT := 0;
	i : USINT := 0;
	pUserData : REFERENCE TO UserDataTyp;
END_VAR
```

#### Main.st
```iecst
PROGRAM _INIT
    // size of Vis structure - this value has to be entered in B&R scene viewer (PVI -> Options -> Size)
	SizeofVis := SIZEOF(Vis);
	// max number of displayed shuttles
	NumVisShuttle := SIZEOF(Vis.Shuttle) / SIZEOF(Vis.Shuttle[0]);
END_PROGRAM

PROGRAM _CYCLIC
	FOR i:=0 TO (NumVisShuttle-1) DO
		IF gShuttleMon.Shuttle[i].Available THEN
			// format selected monitor data to fit B&R scene viewer
			Vis.Shuttle[i].Available     := 1;
			Vis.Shuttle[i].PositionX     := LREAL_TO_REAL(gShuttleMon.Shuttle[i].Position.X);
			Vis.Shuttle[i].PositionY     := LREAL_TO_REAL(gShuttleMon.Shuttle[i].Position.Y);
			Vis.Shuttle[i].RotationZ     := LREAL_TO_REAL(gShuttleMon.Shuttle[i].Orientation.Angle1);
			Vis.Shuttle[i].ExtentToFront := LREAL_TO_REAL(gShuttleMon.Shuttle[i].ExtentToFront);
			Vis.Shuttle[i].ExtentToBack  := LREAL_TO_REAL(gShuttleMon.Shuttle[i].ExtentToBack);
			Vis.Shuttle[i].Width         := LREAL_TO_REAL(gShuttleMon.Shuttle[i].Width);
			//brsitoa(gShuttleMon.Shuttle[i].Index, ADR(Vis.Shuttle[i].Text));
			IF gShuttleMon.Shuttle[i].UserData <> 0 THEN
				pUserData ACCESS gShuttleMon.Shuttle[i].UserData;    // access to user data of this shuttle
				IF pUserData.Color = ORANGE THEN                     // Color is defined with RGB values between 0 and 1
					Vis.Shuttle[i].ColorRed     := 1.000;
					Vis.Shuttle[i].ColorGreen   := 0.5451;
					Vis.Shuttle[i].ColorBlue    := 0.000;
				ELSIF pUserData.Color = GREEN THEN
					Vis.Shuttle[i].ColorRed     := 0.000;
					Vis.Shuttle[i].ColorGreen   := 1.000;
					Vis.Shuttle[i].ColorBlue    := 0.000;
				ELSIF pUserData.Color = RED THEN
					Vis.Shuttle[i].ColorRed     := 1.000;
					Vis.Shuttle[i].ColorGreen   := 0.000;
					Vis.Shuttle[i].ColorBlue    := 0.000;
				ELSIF pUserData.Color = BLUE THEN
					Vis.Shuttle[i].ColorRed     := 0.000;
					Vis.Shuttle[i].ColorGreen   := 0.000;
					Vis.Shuttle[i].ColorBlue    := 1.000;
				ELSIF pUserData.Color = GRAY THEN
					Vis.Shuttle[i].ColorRed     := 0.500;
					Vis.Shuttle[i].ColorGreen   := 0.500;
					Vis.Shuttle[i].ColorBlue    := 0.500;
				ELSIF pUserData.Color = YELLOW THEN
					Vis.Shuttle[i].ColorRed     := 1.000;
					Vis.Shuttle[i].ColorGreen   := 1.000;
					Vis.Shuttle[i].ColorBlue    := 0.000;
				END_IF
			END_IF

		ELSE
			brsmemset(ADR(Vis.Shuttle[i]), 0, SIZEOF(Vis.Shuttle[0]));
		END_IF
	END_FOR
END_PROGRAM

PROGRAM _EXIT
	(* Insert code here *)

END_PROGRAM
```

Listed in the project but not available here: Logical/Global.typ
